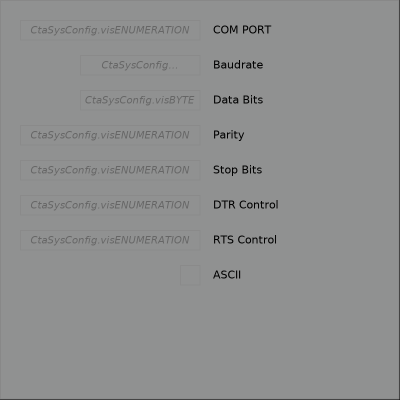
VISUALIZATION VIS_CLIENT_MANAGER_PARAMETER  // 400x400
VAR_INPUT
	ITF_CLIENT_MANAGER_IN : ITF_MB_CLIENTMANAGER;	
END_VAR
    Rectangle (0,0 400x400)
    Frame (0,0 400x400)
        shows VIS_CLIENT_MANAGER_PARAMETER_TCP(ITF_CLIENT_MANAGER_IN := ITF_CLIENT_MANAGER_IN)
    Frame (0,0 400x400)
        shows VIS_CLIENT_MANAGER_PARAMETER_RTU(ITF_CLIENT_MANAGER_IN := ITF_CLIENT_MANAGER_IN)
END_VISUALIZATION

// 40 Visualizations/CLIENTMANAGER/OVERWIEV/VIS_CLIENT_MANAGER_OVERWIEV
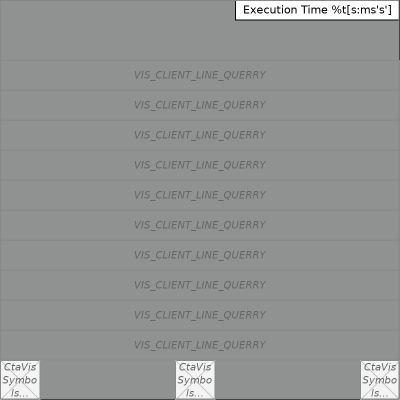
VISUALIZATION VIS_CLIENT_MANAGER_OVERWIEV  // 400x400
VAR_INPUT
	ITF_CLIENT_MANAGER_IN : ITF_MB_CLIENTMANAGER;
END_VAR
    Frame (0,0 400x400), invisible if: NOT __QUERYINTERFACE(ITF_CLIENT_MANAGER_IN,ITF_CLIENT_MANAGER_IN)
        shows VIS_CLIENT_MANAGER_OVERWIEV_QUERRY(ITF_CLIENT_MANAGER_IN := ITF_CLIENT_MANAGER_IN)
END_VISUALIZATION

// 40 Visualizations/CLIENTMANAGER/TCP/PARAMETER/VIS_CLIENT_MANAGER_PARAMETER_TCP
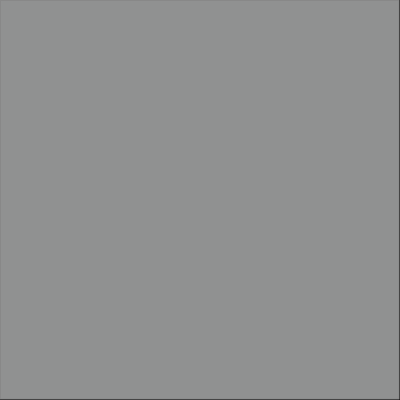
VISUALIZATION VIS_CLIENT_MANAGER_PARAMETER_TCP  // 400x400
VAR_INPUT
	ITF_CLIENT_MANAGER_IN : ITF_MB_CLIENTMANAGER;	
END_VAR
VAR
	ITF_CLIENT_MANAGER_TCP_IN : ITF_MB_CLIENTMANAGER_TCP;	
END_VAR
    Frame (0,0 400x400), invisible if: NOT __QUERYINTERFACE(ITF_CLIENT_MANAGER_IN,ITF_CLIENT_MANAGER_TCP_IN)
        shows VIS_CLIENT_MANAGER_PARAMETER_TCP_QUERY(ITF_CLIENT_MANAGER_TCP_IN := ITF_CLIENT_MANAGER_TCP_IN)
END_VISUALIZATION

// 40 Visualizations/CLIENTMANAGER/TCP/PARAMETER/VIS_CLIENT_MANAGER_PARAMETER_TCP_QUERY
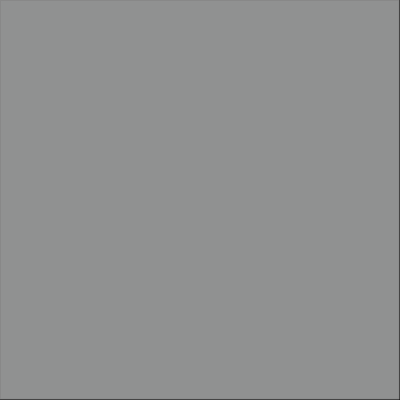
VISUALIZATION VIS_CLIENT_MANAGER_PARAMETER_TCP_QUERY  // 400x400
VAR_INPUT
	ITF_CLIENT_MANAGER_TCP_IN : ITF_MB_CLIENTMANAGER_TCP;	
END_VAR
    Rectangle (0,0 400x400)
END_VISUALIZATION

// 40 Visualizations/CLIENTMANAGER/RTU/PARAMETER/VIS_CLIENT_MANAGER_PARAMETER_RTU
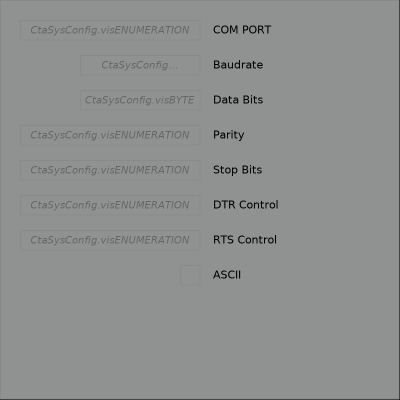
VISUALIZATION VIS_CLIENT_MANAGER_PARAMETER_RTU  // 400x400
VAR_INPUT
	ITF_CLIENT_MANAGER_IN : ITF_MB_CLIENTMANAGER;	
END_VAR
VAR
	ITF_CLIENT_MANAGER_RTU_IN : ITF_MB_CLIENTMANAGER_RTU;	
END_VAR
    Frame (0,0 400x400), invisible if: NOT __QUERYINTERFACE(ITF_CLIENT_MANAGER_IN,ITF_CLIENT_MANAGER_RTU_IN)
        shows VIS_CLIENT_MANAGER_PARAMETER_RTU_QUERY(ITF_CLIENT_MANAGER_RTU_IN := ITF_CLIENT_MANAGER_RTU_IN)
END_VISUALIZATION

// 40 Visualizations/CLIENTMANAGER/RTU/PARAMETER/VIS_CLIENT_MANAGER_PARAMETER_RTU_QUERY
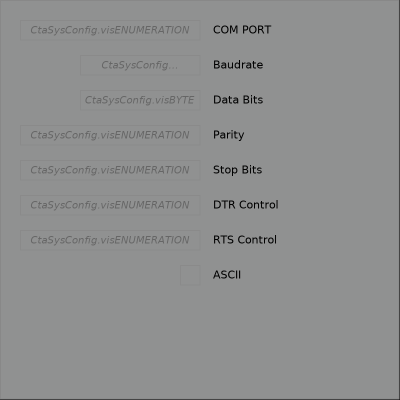
VISUALIZATION VIS_CLIENT_MANAGER_PARAMETER_RTU_QUERY  // 400x400
VAR_INPUT
	ITF_CLIENT_MANAGER_RTU_IN : ITF_MB_CLIENTMANAGER_RTU;	
END_VAR
    Rectangle (0,0 400x400)
    Frame (20,20 180x20), text list: 'TXT_COMPORT', text index: ITF_CLIENT_MANAGER_RTU_IN.P_fbenPort.proValue
        shows CtaSysConfig.visENUMERATION(visfbENUIn := ITF_CLIENT_MANAGER_RTU_IN.P_fbenPort)
    Label (210,20 150x20), "COM PORT"
    Label (210,55 150x20), "Baudrate"
    Frame (80,55 120x20)
        shows CtaSysConfig.visWORD_DEZ(visfbWORDIn := ITF_CLIENT_MANAGER_RTU_IN.P_fbdwBaudrate)
    Label (210,90 150x20), "Data Bits"
    Frame (80,90 120x20)
        shows CtaSysConfig.visBYTE(visfbBYTEIn := ITF_CLIENT_MANAGER_RTU_IN.P_fbbyDataBits)
    Label (210,125 150x20), "Parity"
    Frame (20,125 180x20), text list: 'TXT_COMPORT', text index: ITF_CLIENT_MANAGER_RTU_IN.P_fbenParity.proValue
        shows CtaSysConfig.visENUMERATION(visfbENUIn := ITF_CLIENT_MANAGER_RTU_IN.P_fbenParity)
    Label (210,160 150x20), "Stop Bits"
    Frame (20,160 180x20), text list: 'TEXT_STOPBITS', text index: ITF_CLIENT_MANAGER_RTU_IN.P_fbenStopBits.proValue
        shows CtaSysConfig.visENUMERATION(visfbENUIn := ITF_CLIENT_MANAGER_RTU_IN.P_fbenStopBits)
    Label (210,195 150x20), "DTR Control"
    Frame (20,195 180x20), text list: 'TEXT_DTR_CONTROL', text index: ITF_CLIENT_MANAGER_RTU_IN.P_fbenDTRControl.proValue
        shows CtaSysConfig.visENUMERATION(visfbENUIn := ITF_CLIENT_MANAGER_RTU_IN.P_fbenDTRControl)
    Frame (20,230 180x20), text list: 'TEXT_RTS_CONTROL', text index: ITF_CLIENT_MANAGER_RTU_IN.P_fbenRTSControl.proValue
        shows CtaSysConfig.visENUMERATION(visfbENUIn := ITF_CLIENT_MANAGER_RTU_IN.P_fbenRTSControl)
    Label (210,230 150x20), "RTS Control"
    Frame (180,265 20x20)
        shows CtaSysConfig.visBOOL(visfbBOOLIn := ITF_CLIENT_MANAGER_RTU_IN.P_fbxRtuAscii)
    Label (210,265 150x20), "ASCII"
END_VISUALIZATION

// 40 Visualizations/SERVER/DIA_SERVER
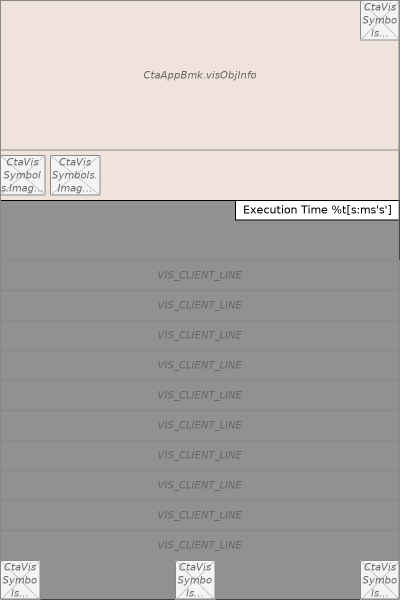
VISUALIZATION DIA_SERVER  // 400x600
VAR_INPUT
	ITF_CLIENT_MANAGER_IN : ITF_MB_CLIENTMANAGER;
END_VAR
VAR
	uiPopUpGruppe 			:	UINT;
END_VAR
    Rectangle (0,0 400x600)
    Frame (0,200 400x400), invisible if: NOT __QUERYINTERFACE(ITF_CLIENT_MANAGER_IN,ITF_CLIENT_MANAGER_IN), frame switch variable: uiPopUpGruppe
        shows VIS_CLIENT_MANAGER_OVERWIEV(ITF_CLIENT_MANAGER_IN := ITF_CLIENT_MANAGER_IN)
        shows VIS_CLIENT_MANAGER_PARAMETER(ITF_CLIENT_MANAGER_IN := ITF_CLIENT_MANAGER_IN)
    Image (360,0 40x40), image: CtaVisSymbols.ImagePool.close_solo_black
        OnMouseClick:  Dialog=Current Dialog, Result=OK, NumpadKeypadSet=True
    Frame (0,155 400x40)
        shows VIS_CLIENTMANAGER_MENÜ(uiPopUpGruppe := uiPopUpGruppe)
    Frame (0,0 400x150)
        shows CtaAppBmk.visObjInfo()
END_VISUALIZATION

// 40 Visualizations/CLIENT/TCP/PARAMETER/VIS_CLIENT_PARAMETER_TCP_TEMP
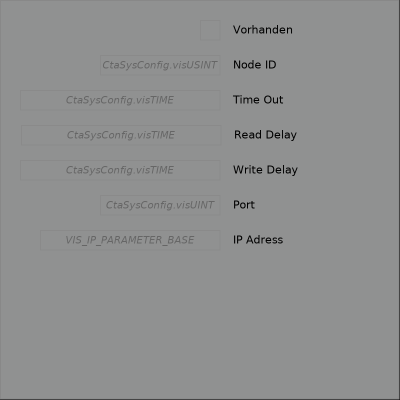
VISUALIZATION VIS_CLIENT_PARAMETER_TCP_TEMP  // 400x400
VAR_INPUT
	ITF_MB_CLIENT_TCP_QUERY	:	ITF_MB_CLIENT_TCP;
END_VAR
    Frame (0,0 400x400), invisible if: NOT __QUERYINTERFACE(ITF_MB_CLIENT_TCP_QUERY,ITF_MB_CLIENT_TCP_QUERY)
        shows VIS_CLIENT_PARAMETER_TCP_QUERY(ITF_MB_CLIENT_TCP_IN := ITF_MB_CLIENT_TCP_QUERY)
END_VISUALIZATION

// 40 Visualizations/CLIENT/RTU/PARAMETER/VIS_CLIENT_PARAMETER_RTU_TEMP
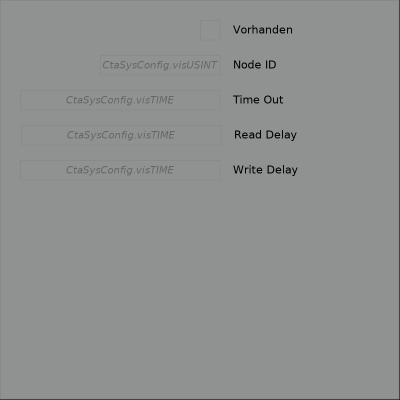
VISUALIZATION VIS_CLIENT_PARAMETER_RTU_TEMP  // 400x400
VAR_INPUT
	ITF_MB_CLIENT_RTU_QUERY	:	ITF_MB_CLIENT_RTU;
END_VAR
    Frame (0,0 400x400), invisible if: NOT __QUERYINTERFACE(ITF_MB_CLIENT_RTU_QUERY,ITF_MB_CLIENT_RTU_QUERY)
        shows VIS_CLIENT_PARAMETER_RTU_QUERY(ITF_MB_CLIENT_RTU_IN := ITF_MB_CLIENT_RTU_QUERY)
END_VISUALIZATION

(* text list txtPhysikalLayer (id | default)
  0 | Default
  1 | RS232
  2 | RS422
  3 | RS423
  4 | RS485 half duplex
  5 | RS485 full duplex
  6 | DMX half duplex
   |  *)

(* text list txtParity (id | default)
  0 | Default
  1 | None
  2 | Odd
  3 | Even
  4 | Mark
  5 | Space
   |  *)

(* text list txtHandshake (id | default)
  0 | Default
  1 | None
  2 | XON XOFF
  3 | DTE RTS CTS
  4 | DCE RTS CTS
  5 | DTE DSR DTR
  6 | DCE DSR DTR
  7 | RTS Lead Time
   |  *)

(* text list txtStopBits (id | default)
  0 | Default
  1 | None
  2 | Minimum
  3 | One
  4 | OneDotFive
  5 | Two
  255 | Maximum
   |  *)

(* text list TEXT_DTR_CONTROL (id | default)
  0 | DTR DISABLE
  1 | DTR ENABLE
  2 | DTR HANDSHAKE
   |  *)

(* text list TEXT_RTS_CONTROL (id | default)
  0 | RTS DISABLE
  1 | RTS ENABLE
  2 | RTS HANDSHAKE
  3 | RTS TOGGLE
   |  *)

(* text list TEXT_STOPBITS (id | default)
  1 | ONE
  2 | ONE DOT FIVE
  3 | TWO
   |  *)

(* text list TXT_COMPORT (id | default)
  0 | NONE
  1 | COM1
  2 | COM2
  3 | COM3
  4 | COM4
   |  *)
